TYPE ST_SavedPositions :
STRUCT
	target		:	REAL;
	description	:	STRING;
	targetclear	:	BOOL:=FALSE;
END_STRUCT
END_TYPE

(* stored: Version 1.1.0.1, ProductVersion 3.1.4022.12
   DUT ST_SavedPositions: Id {07aeed1f-2470-45ab-85fb-9b13cd19d31b} *)
